// TIA Portal V18 export
DATA_BLOCK "Interface"   // DB4
// stored: Access Published, MemoryReserve 100, Namespace nsConvoyeur
   VAR
      "iStart/Stop" : Bool;
      iAccelerate : Bool;
      iDecelerate : Bool;
      ioPosition : UDInt;
      iVitesseRPM : UDInt;
      oVitessePercent : UDInt;
   END_VAR
BEGIN
END_DATA_BLOCK
